% RSLogix 500 project MicroLogix_1100_driver_of Micro8xx_2080-MOT-HSC.RSS, saved by version 8.30.00.16 %
PROJECT "UNTITLED"    % processor: Bul.1763 MicroLogix 1100 Series B %

PROGRAM FILES
  LAD 2   3 rungs

DATA FILES
  O0 OUTPUT  4 elements
  I1 INPUT  6 elements
  S2 STATUS  66 elements
  B3 BINARY  1 elements
  T4 TIMER  4 elements
  C5 COUNTER  1 elements
  R6 CONTROL  1 elements
  N7 INTEGER  1 elements
  F8 FLOAT  1 elements

LADDER 2
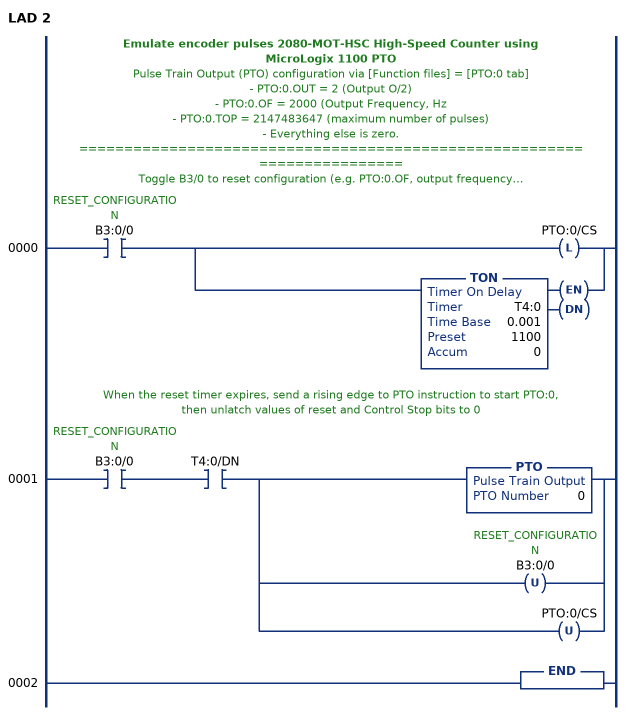
% Rung: 0 %
% TITLE: Emulate encoder pulses 2080-MOT-HSC High-Speed Counter using MicroLogix 1100 PTO %
% Pulse Train Output (PTO) configuration via [Function files] = [PTO:0 tab]
% - PTO:0.OUT = 2 (Output O/2)
% - PTO:0.OF = 2000 (Output Frequency, Hz
% - PTO:0.TOP = 2147483647 (maximum number of pulses)
% - Everything else is zero.
% ========================================================================
% 
% Toggle B3/0 to reset configuration (e.g. PTO:0.OF, output frequency)
% - Latches the value of PTO:0.CS (Control Stop) to 1, which stops PTO
% - Wait 2s after that, then see next rung %
SOR XIC B3:0/0 BST OTL PTO:0/CS NXB TON T4:0 0.001 1100 0 BND EOR
%   B3:0/0  RESET_CONFIGURATION %
% Rung: 1 %
% When the reset timer expires, send a rising edge to PTO instruction to start PTO:0,
% then unlatch values of reset and Control Stop bits to 0 %
SOR XIC B3:0/0 XIC T4:0/DN BST PTO 0 NXB OTU B3:0/0 NXB OTU PTO:0/CS BND EOR
%   B3:0/0  RESET_CONFIGURATION %
% Rung: 2 %
SOR END EOR

DATA TABLE (non-zero values as saved)
DATA T4
% .PRE .ACC %
% T4:0 % 1100 0
% T4:1 % 51 0
% T4:2 % 2560 0
% T4:3 % 5120 0
DATA C5
% .PRE .ACC %
% C5:0 % 6001 0
